// TIA Portal V19 export
DATA_BLOCK "LB113_W"   // DB90
// stored: InstanceOfName ButtonsSafe_LB113_W, InstanceOfType FB
"ButtonsSafe_LB113_W"
   // VAR_INPUT
   //    Reset_OthersPBs_Activation_IN : Bool;
   // END_VAR
   // VAR_OUTPUT
   //    Reset_OthersPBs_Activation_OUT : Bool;
   // END_VAR
   // VAR
   //    i : Int;
   //    iOperation : Int;
   //    iConcurrentOperation : Int;
   //    SettingWriteDone : Bool;
   //    PbPanel : "Buttons2Hands";
   //    PB : Struct
   //       ResetAlarms : Bool;
   //       JBTorch_Fwd : Bool;
   //       JBTorch_Bwd : Bool;
   //       JBWeldMan : Bool;
   //    END_STRUCT;
   // END_VAR
BEGIN
END_DATA_BLOCK
